// TIA Portal V19 export
TYPE "LAF_typeAxisDiagStatusWord2"
TITLE = LAF_typeAxisDiagStatusWord2
// Status information of a Technology object
// stored: Access Published
   STRUCT
      bit00_StopCommand { ExternalWritable := 'False'} : Bool;   // An "MC_Stop" job is running. The technology object is disabled / Enable
      bit01_DesynchronizingCommand { ExternalWritable := 'False'} : Bool;   // An "MC_GearOut" job or "MC_CamOut" job is active. The following axis is desynchronized / Error
      bit02_PassingBacklash { ExternalWritable := 'False'} : Bool;   // The backlash is traversed. "<TO>.ActualPosition" does not hereby change / RestartActive
      bit03_PhasingCommandWaiting { ExternalWritable := 'False'} : Bool;   // An "MC_PhasingAbsolute" or "MC_PhasingRelative" job for leading value offset is waiting / OnlineStartValuesChanged
      bit04_OffsetCommand { ExternalWritable := 'False'} : Bool;   // An "MC_OffsetAbsolute" or "MC_OffsetRelative" job for following value offset is active / ControlPanelActive
      bit05_OffsetCommandWaiting { ExternalWritable := 'False'} : Bool;   // An "MC_OffsetAbsolute" or "MC_OffsetRelative" job for following value offset is waiting / HomingDone
      bit06_MotionInSuperimposedCommand { ExternalWritable := 'False'} : Bool;   // An "MC_MotionInSuperimposed" job is running / Done
      bit07_HaltSuperimposedCommand { ExternalWritable := 'False'} : Bool;   // An "MC_HaltSuperimposed" job is running / StandStill
      bit08_Reserved { ExternalWritable := 'False'} : Bool;   // Reserved / PositioningCommand
      bit09_Reserved { ExternalWritable := 'False'} : Bool;   // Reserved / JogCommand
      bit10_Reserved { ExternalWritable := 'False'} : Bool;   // Reserved / VelocityCommand
      bit11_Reserved { ExternalWritable := 'False'} : Bool;   // Reserved / HomingCommand
      bit12_Reserved { ExternalWritable := 'False'} : Bool;   // Reserved / ConstantVelocity
      bit13_Reserved { ExternalWritable := 'False'} : Bool;   // Reserved / Accelerating
      bit14_Reserved { ExternalWritable := 'False'} : Bool;   // Reserved / Decelerating
      bit15_Reserved { ExternalWritable := 'False'} : Bool;   // Reserved / SWLimitMinActive
      bit16_Reserved { ExternalWritable := 'False'} : Bool;   // Reserved / SWLimitMaxActive
      bit17_Reserved { ExternalWritable := 'False'} : Bool;   // Reserved / HWLimitMinActive
      bit18_Reserved { ExternalWritable := 'False'} : Bool;   // Reserved / HWLimitMaxActive
      bit19_Reserved { ExternalWritable := 'False'} : Bool;   // Reserved
      bit20_Reserved { ExternalWritable := 'False'} : Bool;   // Reserved
      bit21_Reserved { ExternalWritable := 'False'} : Bool;   // Reserved / Synchronizing
      bit22_Reserved { ExternalWritable := 'False'} : Bool;   // Reserved / Synhronous
      bit23_Reserved { ExternalWritable := 'False'} : Bool;   // Reserved / SuperimposedMotionCommand
      bit24_Reserved { ExternalWritable := 'False'} : Bool;   // Reserved / PhasingCommand
      bit25_Reserved { ExternalWritable := 'False'} : Bool;   // Reserved / AxisSimulation
      bit26_Reserved { ExternalWritable := 'False'} : Bool;   // Reserved / TorqueLimitingCommand
      bit27_Reserved { ExternalWritable := 'False'} : Bool;   // Reserved / InLimitation
      bit28_Reserved { ExternalWritable := 'False'} : Bool;   // Reserved / NonPositionControlled
      bit29_Reserved { ExternalWritable := 'False'} : Bool;   // Reserved
      bit30_Reserved { ExternalWritable := 'False'} : Bool;   // Reserved / InClamping
      bit31_Reserved { ExternalWritable := 'False'} : Bool;   // Reserved
   END_STRUCT;
END_TYPE
